// Mitsubishi GX Works2 project: 0630   PLC: Q03UDV

// global labels: Global1
VAR_GLOBAL
  공급후진리드 AT X20 : BOOL;
  공급전진리드 AT X21 : BOOL;
  매거진센서 AT X22 : BOOL;
  고주파센서 AT X23 : BOOL;
  용량형센서 AT X24 : BOOL;
  근접포토센서 AT X25 : BOOL;
  그리퍼온리드 AT X27 : BOOL;
  그리퍼오프리드 AT X28 : BOOL;
  물품도착포토 AT X29 : BOOL;
  TG1 AT X2A : BOOL;
  TG2 AT X2B : BOOL;
  TG3 AT X2C : BOOL;
  PB4 AT X2D : BOOL;
  PB5 AT X2E : BOOL;
  창고1 AT X30 : BOOL;
  창고2 AT X31 : BOOL;
  창고3 AT X32 : BOOL;
  창고4 AT X33 : BOOL;
  창고5 AT X34 : BOOL;
  창고6 AT X35 : BOOL;
  창고7 AT X36 : BOOL;
  창고8 AT X37 : BOOL;
  창고9 AT X38 : BOOL;
  도어센서 AT X39 : BOOL;
  압력센서 AT X3A : BOOL;
  공급전솔 AT Y40 : BOOL;
  공급후솔 AT Y41 : BOOL;
  그리퍼온솔 AT Y42 : BOOL;
  그리퍼오프솔 AT Y43 : BOOL;
  경광녹색 AT Y44 : BOOL;
  경광황색 AT Y45 : BOOL;
  경광적색 AT Y46 : BOOL;
  부저 AT Y47 : BOOL;
  컨베이어 AT Y48 : BOOL;
  램프1 AT Y4A : BOOL;
  램프2 AT Y4B : BOOL;
  램프3 AT Y4C : BOOL;
  램프5 AT Y4D : BOOL;
  램프4 AT Y4E : BOOL;
  R그립온명령 AT X1000 : BOOL;
  R그립오프명령 AT X1001 : BOOL;
  R_PLC시작 AT X1002 : BOOL;
  R_판별리셋 AT X1003 : BOOL;
  R재공급 AT X1004 : BOOL;
  R그립온센서 AT Y1000 : BOOL;
  R그립오프센서 AT Y1001 : BOOL;
  R물품없음 AT Y1002 : BOOL;
  R_금속 AT Y1003 : BOOL;
  R_검비금속 AT Y1004 : BOOL;
  R_흰비금속 AT Y1005 : BOOL;
  R물품도착 AT Y1006 : BOOL;
  R컨베이어 AT Y1007 : BOOL;
  R_재시작 AT Y1008 : BOOL;
  R_interrupt AT Y1009 : BOOL;
  R창고1 AT Y100A : BOOL;
  R창고2 AT Y100B : BOOL;
  R창고3 AT Y100C : BOOL;
  R창고4 AT Y100D : BOOL;
  R창고5 AT Y100E : BOOL;
  R창고6 AT Y100F : BOOL;
  R창고7 AT Y1010 : BOOL;
  R창고8 AT Y1011 : BOOL;
  R창고9 AT Y1012 : BOOL;
  R창고A AT Y1013 : BOOL;
END_VAR

PROGRAM MAIN
VAR
  T_매거진없음 : TIMER;
  공작물공급 : BOOL;
  작동중 : BOOL;
  비화 : BOOL;
  비금 : BOOL;
  금속 : BOOL;
  T_컨베이어 : TIMER;
  종료 : BOOL;
  컨정지 : BOOL;
END_VAR
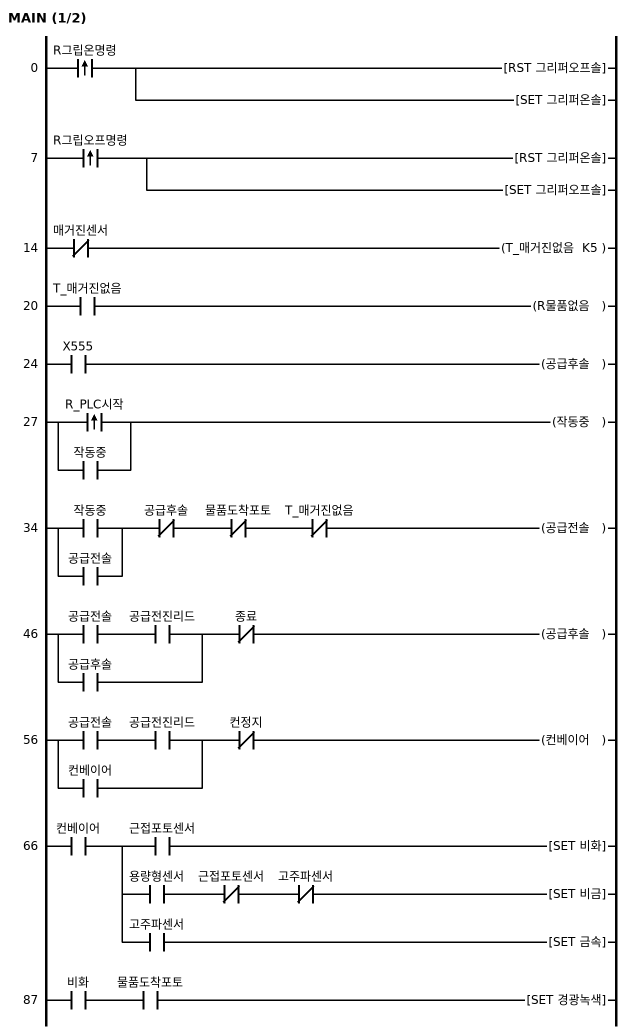
0     LDP     R그립온명령
      RST     그리퍼오프솔
      SET     그리퍼온솔
7     LDP     R그립오프명령
      RST     그리퍼온솔
      SET     그리퍼오프솔
14    LDI     매거진센서
      OUT     T_매거진없음 K5
20    LD      T_매거진없음
      OUT     R물품없음
24    LD      X555
      OUT     공급후솔
27    LDP     R_PLC시작
      OR      작동중
      OUT     작동중
34    LD      작동중
      OR      공급전솔
      ANI     공급후솔
      ANI     물품도착포토
      ANI     T_매거진없음
      OUT     공급전솔
46    LD      공급전솔
      AND     공급전진리드
      OR      공급후솔
      ANI     종료
      OUT     공급후솔
56    LD      공급전솔
      AND     공급전진리드
      OR      컨베이어
      ANI     컨정지
      OUT     컨베이어
66    LD      컨베이어
      MPS
      AND     근접포토센서
      SET     비화
      MRD
      AND     용량형센서
      ANI     근접포토센서
      ANI     고주파센서
      SET     비금
      MPP
      AND     고주파센서
      SET     금속
87    LD      비화
      AND     물품도착포토
      SET     경광녹색
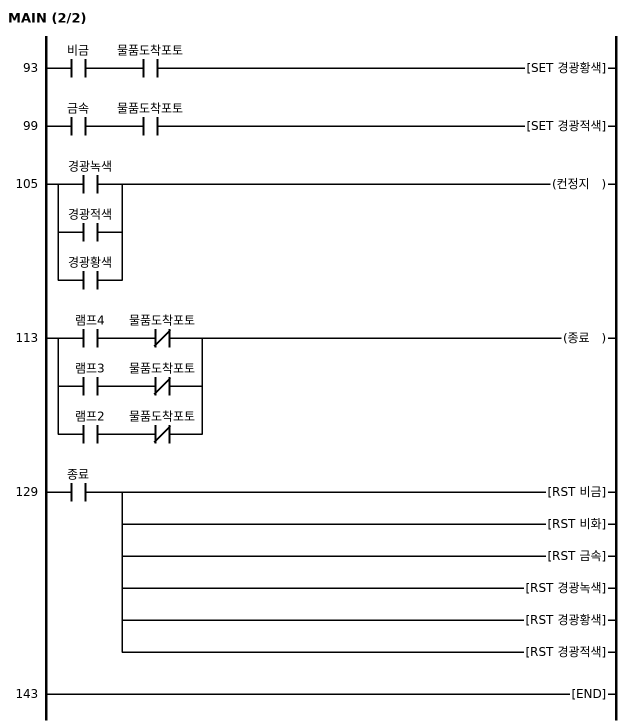
93    LD      비금
      AND     물품도착포토
      SET     경광황색
99    LD      금속
      AND     물품도착포토
      SET     경광적색
105   LD      경광녹색
      OR      경광적색
      OR      경광황색
      OUT     컨정지
113   LD      램프4
      ANI     물품도착포토
      LD      램프3
      ANI     물품도착포토
      ORB
      LD      램프2
      ANI     물품도착포토
      ORB
      OUT     종료
129   LD      종료
      RST     비금
      RST     비화
      RST     금속
      RST     경광녹색
      RST     경광황색
      RST     경광적색
143   END
END_PROGRAM
